# EPICS autosave request: ADApp/Db/ADFile_settings.req
$(P)$(F)BlockingCallbacks
$(P)$(F)FilePath
$(P)$(F)FileName
$(P)$(F)FileNumber
$(P)$(F)AutoIncrement
$(P)$(F)FileTemplate
$(P)$(F)AutoSave
$(P)$(F)FileFormat
$(P)$(F)FileWriteMode
$(P)$(F)NumCapture
